(* PLC project Unnamed, Unknown Unnamed 1 *)
(* stored: creationDateTime 2023-04-26T09:18:19, modificationDateTime 2023-05-25T11:47:17 *)

PROGRAM OPLC_SORTBYMOD2
  VAR
    ATENTRY : BOOL;
    ATBACK : BOOL;
    LOWBOX : BOOL;
    HIGHBOX : BOOL;
    TURNTABLEENTRY : BOOL;
    LOADPOS : BOOL;
    UNLOADPOS : BOOL;
    ATFRONT : BOOL;
    RIGHTENT : BOOL;
    LEFTENT : BOOL;
    RIGHTEXIT : BOOL;
    LEFTEXIT : BOOL;
    START : BOOL;
    RESET : BOOL;
    STOP : BOOL;
    EMERGENCY : BOOL;
    MACH_ON : BOOL;
    MACH_OFF : BOOL;
    FEEDERCONV : BOOL;
    ENTRYCONV : BOOL;
    LOAD : BOOL;
    UNLOAD : BOOL;
    TURN : BOOL;
    LEFTCONV : BOOL;
    RIGHTCONV : BOOL;
    GREENIND : BOOL;
    YELLOWIND : BOOL;
    REDIND : BOOL;
    LSTART : BOOL;
    LRESET : BOOL;
    LSTOP : BOOL;
    CONT : BOOL;
    CONTINUERIGHT : BOOL;
    CONTINUELEFT : BOOL;
    ET : TIME;
    PV : WORD;
    CV : WORD;
    MEMOLEFT : BOOL;
    MEMORIGHT : BOOL;
    UNTURN : BOOL;
    TOF0 : TOF;
  END_VAR

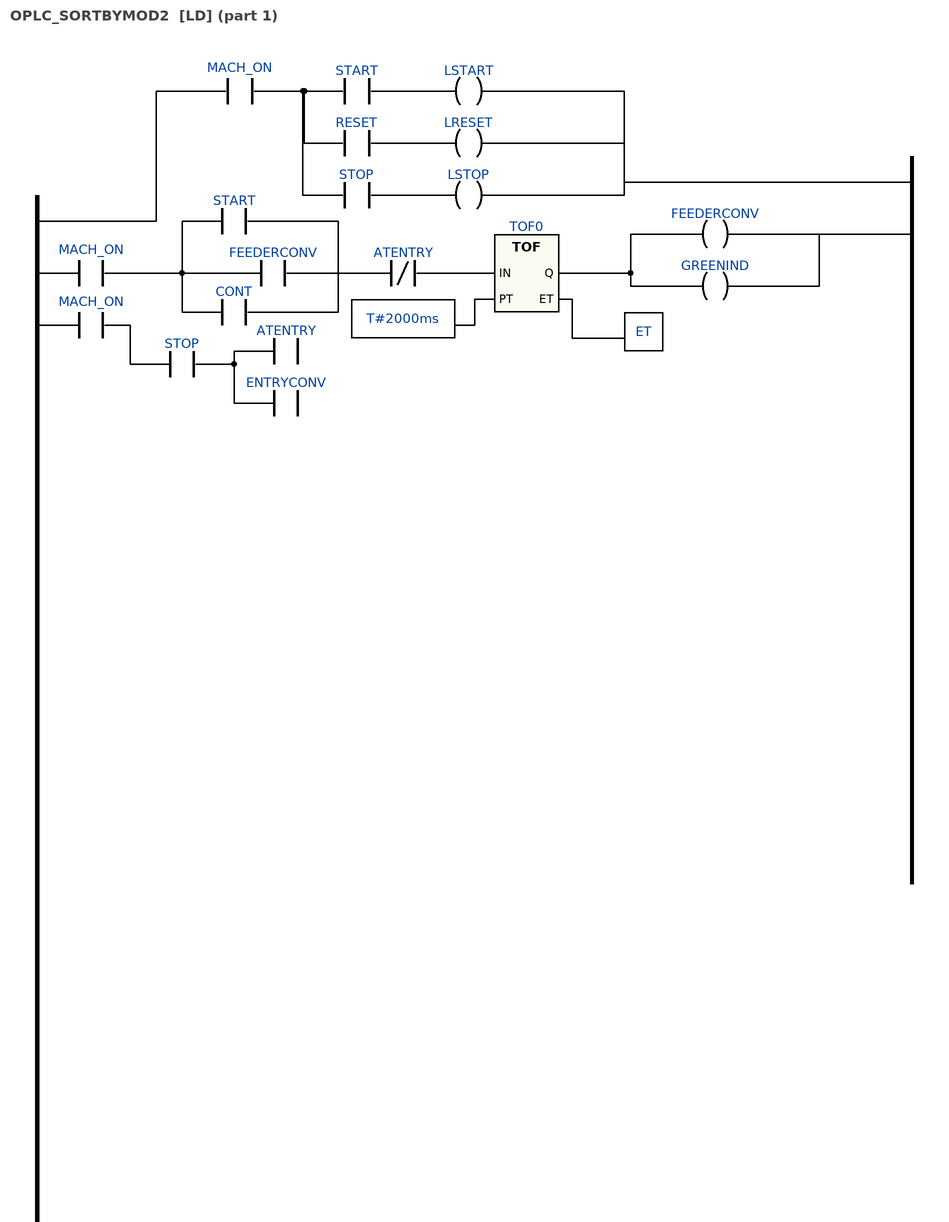
(* LD diagram, written out as Structured Text *)
LSTART := MACH_ON AND START;
LRESET := MACH_ON AND RESET;
LSTOP := MACH_ON AND STOP;
TOF0(IN := MACH_ON AND (FEEDERCONV OR CONT OR START) AND NOT ATENTRY, PT := T#2000ms);
FEEDERCONV := TOF0.Q;
GREENIND := TOF0.Q;
ET := TOF0.ET;
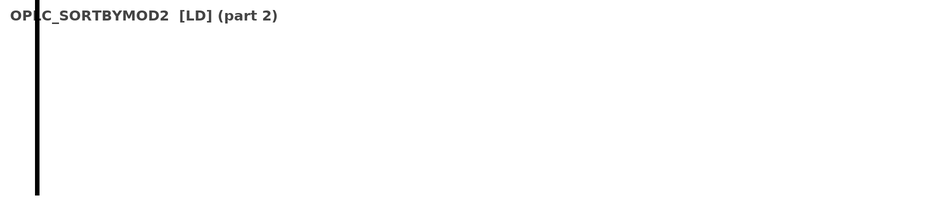
(* drawn but not wired to any output: MACH_ON, STOP, ATENTRY, ENTRYCONV *)
END_PROGRAM

CONFIGURATION Config0
  RESOURCE Res0 ON PLC
    TASK task0(INTERVAL := T#20ms, PRIORITY := 0);
    PROGRAM instance0 WITH task0 : OPLC_SORTBYMOD2;
  END_RESOURCE
END_CONFIGURATION
